(*
SPDX-FileCopyrightText: Â© 2026 Oleksandr Tiutyk <trofimich@gmail.com>
SPDX-License-Identifier: MIT
License: https://opensource.org/license/mit
*)

(*!
<summary>Identifies underlying data type of a raw ADC or DAC analog signal.</summary>
<description>
Specifies whether the raw process data is interpreted as signed 16-bit integer, signed 32-bit integer,
or 32-bit single-precision floating point.
</description>
*)

{attribute 'qualified_only'}
{attribute 'strict'}
{attribute 'to_string'}
TYPE RAW_ANALOG_VALUE_TYPE :
(
	INT16,
	INT32,
	REAL32 
);
END_TYPE

(* stored: Version 1.1.0.1
   DUT RAW_ANALOG_VALUE_TYPE: Id {f2da2152-048b-4bfc-b0b9-1b69bda969dc} *)
